{attribute 'linkalways'}
{attribute 'hide_all_locals'}
FUNCTION_BLOCK ValueRealRead EXTENDS ValueBase IMPLEMENTS ValueRead
VAR
	thisValue : REAL;
END_VAR

{attribute 'call_after_global_init_slot' := '1'}
{attribute 'call_after_online_change_slot' := '1'}
METHOD PROTECTED GetThisAnyType
VAR_INPUT
END_VAR
thisAnyType := ToAnyType(thisValue);
END_METHOD

METHOD GetAsType : BOOL
VAR_INPUT
	destination : __SYSTEM.AnyType;
END_VAR
GetAsType := ConvertAnyType(thisAnyType, destination);
END_METHOD

METHOD GetAsString : T_MaxString
VAR_INPUT
END_VAR
GetAsString := TO_STRING(thisValue);
END_METHOD

METHOD Get : BOOL
VAR_INPUT
	destination : ANY;
END_VAR
Get := ConvertAnyType(thisAnyType, destination);
END_METHOD

METHOD FB_init : BOOL
VAR_INPUT
	bInitRetains : BOOL; // if TRUE, the retain variables are initialized (warm start / cold start)
	bInCopyCode : BOOL;  // if TRUE, the instance afterwards gets moved into the copy code (online change)
END_VAR
_ValueType := __SYSTEM.TYPE_CLASS.TYPE_REAL;
END_METHOD

{attribute 'monitoring' := 'call'}
PROPERTY Value : REAL
GET
Value := thisValue;
END_GET
END_PROPERTY

END_FUNCTION_BLOCK

(* stored: Version 1.1.0.1
   POU ValueRealRead: Id {a45a6aea-0c1b-4f47-828b-0f52577f9584}, SpecialFunc None
   Method GetThisAnyType: Id {eee0ecca-4770-4f27-b505-a0b4995fcb7d}
   Method GetAsType: Id {7b05bcbb-8b43-4a43-a253-4b4faa03baa6}
   Method GetAsString: Id {d8d6eb95-742b-40a0-bb39-bc9af4ed0efa}
   Method Get: Id {f5fd3c88-e038-4192-afc2-fdafc92e307f}
   Method FB_init: Id {a8958567-444f-420b-af81-73e8dceb6771}
   Property Value: Id {84464656-395e-4e11-8da1-b211f166ec16}
   Get Get: Id {1dffb567-0a32-4db0-9e06-64f33bc1478d} *)
